(* IEC 61131-3 sources: Lasal/CPU_5344_V01/Class/CtrlCheckMachineReady, 1 file *)

(* ---- CtrlCheckMachineReady.st ---- *)
(*!
<Class
	Name               = "CtrlCheckMachineReady"
	Revision           = "0.1"
	RealtimeTask       = "false"
	CyclicTask         = "true"
	DefCyclictime      = "50 ms"
	BackgroundTask     = "false"
	Sigmatek           = "false"
	OSInterface        = "false"
	HighPriority       = "false"
	Automatic          = "false"
	UpdateMode         = "Prescan"
	SharedCommandTable = "true"
	Objectsize         = "(570,120)">
	<Channels>
		<Server Name="AlarmActiefCommon" Visualized="true" Initialize="false" WriteProtected="false" Retentive="false"/>
		<Server Name="AlarmActiefSafety" Visualized="true" Initialize="false" WriteProtected="false" Retentive="false"/>
		<Server Name="AlarmLubr" Visualized="true" Initialize="false" WriteProtected="false" Retentive="false"/>
		<Server Name="ClassSvr" Visualized="false" Initialize="false" WriteProtected="true" Retentive="false"/>
		<Server Name="ErrorNrCommon" Visualized="true" Initialize="false" WriteProtected="false" Retentive="false"/>
		<Server Name="ErrorNrLubr" Visualized="true" Initialize="false" WriteProtected="false" Retentive="false"/>
		<Server Name="ErrorNrSafety" Visualized="true" Initialize="false" WriteProtected="false" Retentive="false"/>
		<Server Name="ResetAlarms" Visualized="false" Initialize="false" WriteProtected="false" Retentive="false"/>
		<Server Name="result" Class="Logic_Or_2" Visualized="true" Remotely="true" Initialize="false" WriteProtected="true" Retentive="false" Comment="result of logic operation"/>
		<Server Name="sStartUpTime" Visualized="false" Initialize="true" DefValue="10000" WriteProtected="true" Retentive="false"/>
		<Server Name="Status_Controlcurrent" Visualized="false" Initialize="false" WriteProtected="false" Retentive="false"/>
		<Server Name="Status_SafeCompleet" Visualized="false" Initialize="false" WriteProtected="false" Retentive="false"/>
		<Client Name="_AlarmCommon" Required="true" Internal="true"/>
		<Client Name="_AlarmLubr" Required="true" Internal="true"/>
		<Client Name="_AlarmSafety" Required="true" Internal="true"/>
		<Client Name="iBlink" Required="true" Internal="false"/>
		<Client Name="iBTBs" Required="false" Internal="false"/>
		<Client Name="iControlCurrent" Required="true" Internal="false"/>
		<Client Name="iEmergencyStops" Required="false" Internal="false"/>
		<Client Name="iIsafeCompleet" Required="true" Internal="false"/>
		<Client Name="iLuchtdrukOK" Required="false" Internal="false"/>
		<Client Name="iNrLubrs" Required="false" Internal="false"/>
		<Client Name="iSimulateMode" Required="false" Internal="false"/>
		<Client Name="iSmeerSystemenLeeg" Required="false" Internal="false"/>
		<Client Name="iStatusCanComm" Required="true" Internal="false" DefValue="1"/>
		<Client Name="iStuurstroomIn" Required="false" Internal="false"/>
		<Client Name="iThermUits" Required="false" Internal="false"/>
		<Client Name="Logic_Or_23" Required="true" Internal="true"/>
		<Client Name="Logic_Or_24" Required="true" Internal="true"/>
		<Client Name="nrBTBinUse" Required="false" Internal="false"/>
		<Client Name="nrEmergencyStops" Required="false" Internal="false"/>
		<Client Name="nrThermUitinUse" Required="false" Internal="false"/>
		<Client Name="oLightControlCurrent" Required="false" Internal="false"/>
		<Client Name="StatusIOlinkComm" Required="false" Internal="false"/>
	</Channels>
	<RevDoku>
		<Owner/>
		<Dokumentation Revision="0.1" Date="2021-02-09" Author="JDK&#13;&#10;" Company="Dulst" Description="Add lub alarms&#13;&#10;"/>
	</RevDoku>
	<Network Name="CtrlCheckMachineReady">
		<!-- List of Components in this network -->
		<Components>
			<Object
				Name           = "_AlarmCommon"
				Class          = "_AlarmX3ParaDer"
				Position       = "(600,1110)"
				Visualized     = "true"
				Remotely       = "true"
				BackgroundTime = "100 ms">
				<Channels>
					<Server Name="AlarmActief"/>
					<Server Name="ClassSvr"/>
					<Server Name="ErrorNr"/>
					<Client Name="Acknow"/>
					<Client Name="Config" Value="0"/>
					<Client Name="Group"/>
					<Client Name="Para1"/>
					<Client Name="Para2"/>
					<Client Name="Para3"/>
				</Channels>
			</Object>
			<Object
				Name           = "_AlarmLubr"
				Class          = "_AlarmX3ParaDer"
				Position       = "(630,2100)"
				Visualized     = "true"
				Remotely       = "true"
				BackgroundTime = "100 ms">
				<Channels>
					<Server Name="AlarmActief"/>
					<Server Name="ClassSvr"/>
					<Server Name="ErrorNr"/>
					<Client Name="Acknow"/>
					<Client Name="Config" Value="0"/>
					<Client Name="Group"/>
					<Client Name="Para1"/>
					<Client Name="Para2"/>
					<Client Name="Para3"/>
				</Channels>
			</Object>
			<Object
				Name           = "_AlarmSafety"
				Class          = "_AlarmX3ParaDer"
				Position       = "(600,1620)"
				Visualized     = "true"
				Remotely       = "true"
				BackgroundTime = "100 ms">
				<Channels>
					<Server Name="AlarmActief"/>
					<Server Name="ClassSvr"/>
					<Server Name="ErrorNr"/>
					<Client Name="Acknow"/>
					<Client Name="Config" Value="0"/>
					<Client Name="Group"/>
					<Client Name="Para1"/>
					<Client Name="Para2"/>
					<Client Name="Para3"/>
				</Channels>
			</Object>
			<Object
				Name       = "Logic_Or_23"
				Class      = "Logic_Or_2"
				Position   = "(1530,2310)"
				Visualized = "true"
				Remotely   = "true">
				<Channels>
					<Server Name="Result"/>
					<Client Name="Op1"/>
					<Client Name="Op2"/>
				</Channels>
			</Object>
			<Object
				Name       = "Logic_Or_24"
				Class      = "Logic_Or_2"
				Position   = "(1410,1950)"
				Visualized = "true"
				Remotely   = "true">
				<Channels>
					<Server Name="Result"/>
					<Client Name="Op1"/>
					<Client Name="Op2"/>
				</Channels>
			</Object>
		</Components>
		<Comments>
		</Comments>
		<!-- List of Connections in this network -->
		<Connections>
			<Connection Source="this._AlarmLubr" Destination="_AlarmLubr.ClassSvr"/>
			<Connection Source="this._AlarmCommon" Destination="_AlarmCommon.ClassSvr"/>
			<Connection Source="this.AlarmActiefCommon" Destination="_AlarmCommon.AlarmActief" Vertices="(2002,450),(916,1260),"/>
			<Connection Source="this.ErrorNrCommon" Destination="_AlarmCommon.ErrorNr" Vertices="(2002,630),(916,1320),"/>
			<Connection Source="this._AlarmSafety" Destination="_AlarmSafety.ClassSvr"/>
			<Connection Source="this.AlarmActiefSafety" Destination="_AlarmSafety.AlarmActief" Vertices="(2002,510),(916,1770),"/>
			<Connection Source="this.ErrorNrSafety" Destination="_AlarmSafety.ErrorNr" Vertices="(2002,690),(916,1830),"/>
			<Connection Source="this.AlarmLubr" Destination="_AlarmLubr.AlarmActief" Vertices="(2002,570),(946,2250),"/>
			<Connection Source="this.ErrorNrLubr" Destination="_AlarmLubr.ErrorNr" Vertices="(2002,750),(946,2310),"/>
			<Connection Source="this.Logic_Or_23" Destination="Logic_Or_23.Result"/>
			<Connection Source="this.Logic_Or_24" Destination="Logic_Or_24.Result"/>
			<Connection Source="Logic_Or_24.Op1" Destination="_AlarmCommon.AlarmActief" Vertices="(1410,2040),(916,1260),"/>
			<Connection Source="Logic_Or_24.Op2" Destination="_AlarmSafety.AlarmActief" Vertices="(1410,2100),(916,1770),"/>
			<Connection Source="Logic_Or_23.Op2" Destination="_AlarmLubr.AlarmActief" Vertices="(1530,2460),(946,2250),"/>
			<Connection Source="Logic_Or_23.Op1" Destination="Logic_Or_24.Result" Vertices="(1530,2400),(1710,2040),"/>
			<Connection Source="this.result" Destination="Logic_Or_23.Result" Vertices="(2002,870),(1830,2400),"/>
		</Connections>
		<!-- Headerfiles -->
		<Options>
		</Options>
	</Network>
</Class>
*)
CtrlCheckMachineReady : CLASS
  //Servers:
	ClassSvr 	: SvrChCmd_DINT;
	Status_SafeCompleet 	: SvrCh_DINT;
	Status_Controlcurrent 	: SvrCh_DINT;
	ResetAlarms 	: SvrCh_DINT;
	AlarmActiefCommon 	: SvrCh_DINT;
	AlarmActiefSafety 	: SvrCh_DINT;
	AlarmLubr 	: SvrCh_DINT;
	ErrorNrCommon 	: SvrCh_DINT;
	ErrorNrSafety 	: SvrCh_DINT;
	ErrorNrLubr 	: SvrCh_DINT;
	sStartUpTime 	: SvrCh_UDINT;
	result 	: SvrChCmd_DINT;
  //Clients:
	StatusIOlinkComm 	: CltCh_DINT;
	iStatusCanComm 	: CltCh_DINT;
	iStuurstroomIn 	: CltCh_DINT;
	iBTBs 	: CltChCmd_Lees10Ingangenin;
	nrBTBinUse 	: CltCh_DINT;
	iThermUits 	: CltChCmd_Lees10Ingangenin;
	nrThermUitinUse 	: CltCh_DINT;
	iSmeerSystemenLeeg 	: CltCh_DINT;
	iLuchtdrukOK 	: CltCh_DINT;
	iEmergencyStops 	: CltChCmd_Lees10Ingangenin;
	nrEmergencyStops 	: CltCh_DINT;
	oLightControlCurrent 	: CltCh_DINT;
	iSimulateMode 	: CltCh_eSimuState;
	iIsafeCompleet 	: CltCh_DINT;
	iControlCurrent 	: CltCh_DINT;
	iBlink 	: CltCh_DINT;
	iNrLubrs 	: CltCh_DINT;
	_AlarmCommon 	: CltChCmd__AlarmX3ParaDer;
	_AlarmSafety 	: CltChCmd__AlarmX3ParaDer;
	_AlarmLubr 	: CltChCmd__AlarmX3ParaDer;
	Logic_Or_23 	: CltChCmd_Logic_Or_2;
	Logic_Or_24 	: CltChCmd_Logic_Or_2;
  //Variables:
		i 	: DINT;
		ii 	: DINT;
		tmp 	: DINT;
		Status_OldErrorNr 	: DINT;
		tmpErrorNrCommon 	: DINT;
		tmpErrorNrSafety 	: DINT;
		tmpErrorLubr 	: DINT;
  //Functions:

	FUNCTION VIRTUAL GLOBAL CyWork
		VAR_INPUT
			EAX 	: UDINT;
		END_VAR
		VAR_OUTPUT
			state (EAX) 	: UDINT;
		END_VAR;

	FUNCTION CheckNr
		VAR_INPUT
			nr 	: DINT;
			aantaltoread 	: DINT;
			offset 	: DINT;
		END_VAR
		VAR_OUTPUT
			HighNr 	: DINT;
		END_VAR;

	FUNCTION CheckStStrBTBenTherm;

	FUNCTION PreScan;

	FUNCTION CheckSmeerSysteem;

	FUNCTION giveAlarmCommon
		VAR_INPUT
			errorNr 	: DINT;
		END_VAR;

	FUNCTION giveAlarmSafety
		VAR_INPUT
			errorNr 	: DINT;
		END_VAR;

	FUNCTION VIRTUAL GLOBAL ResetAlarms::Write
		VAR_INPUT
			input (EAX) 	: DINT;
		END_VAR
		VAR_OUTPUT
			result (EAX) 	: DINT;
		END_VAR;

	FUNCTION VIRTUAL GLOBAL AlarmActiefCommon::Read
		VAR_OUTPUT
			output (EAX) 	: DINT;
		END_VAR;

	FUNCTION VIRTUAL GLOBAL AlarmActiefCommon::Write
		VAR_INPUT
			input (EAX) 	: DINT;
		END_VAR
		VAR_OUTPUT
			result (EAX) 	: DINT;
		END_VAR;

	FUNCTION VIRTUAL GLOBAL AlarmActiefSafety::Read
		VAR_OUTPUT
			output (EAX) 	: DINT;
		END_VAR;

	FUNCTION VIRTUAL GLOBAL AlarmActiefSafety::Write
		VAR_INPUT
			input (EAX) 	: DINT;
		END_VAR
		VAR_OUTPUT
			result (EAX) 	: DINT;
		END_VAR;

	FUNCTION VIRTUAL GLOBAL AlarmLubr::Read
		VAR_OUTPUT
			output (EAX) 	: DINT;
		END_VAR;

	FUNCTION VIRTUAL GLOBAL AlarmLubr::Write
		VAR_INPUT
			input (EAX) 	: DINT;
		END_VAR
		VAR_OUTPUT
			result (EAX) 	: DINT;
		END_VAR;

	FUNCTION VIRTUAL GLOBAL ErrorNrCommon::Read
		VAR_OUTPUT
			output (EAX) 	: DINT;
		END_VAR;

	FUNCTION VIRTUAL GLOBAL ErrorNrCommon::Write
		VAR_INPUT
			input (EAX) 	: DINT;
		END_VAR
		VAR_OUTPUT
			result (EAX) 	: DINT;
		END_VAR;

	FUNCTION VIRTUAL GLOBAL ErrorNrSafety::Read
		VAR_OUTPUT
			output (EAX) 	: DINT;
		END_VAR;

	FUNCTION VIRTUAL GLOBAL ErrorNrSafety::Write
		VAR_INPUT
			input (EAX) 	: DINT;
		END_VAR
		VAR_OUTPUT
			result (EAX) 	: DINT;
		END_VAR;

	FUNCTION VIRTUAL GLOBAL ErrorNrLubr::Read
		VAR_OUTPUT
			output (EAX) 	: DINT;
		END_VAR;

	FUNCTION VIRTUAL GLOBAL ErrorNrLubr::Write
		VAR_INPUT
			input (EAX) 	: DINT;
		END_VAR
		VAR_OUTPUT
			result (EAX) 	: DINT;
		END_VAR;

	FUNCTION VIRTUAL GLOBAL result::Read
		VAR_OUTPUT
			output (EAX) 	: DINT;
		END_VAR;
  //Tables:
	FUNCTION @STD
		VAR_OUTPUT
			ret_code	: CONFSTATES;
		END_VAR;
	FUNCTION GLOBAL TAB @CT_;
END_CLASS;

#pragma using _AlarmX3ParaDer
#pragma using Logic_Or_2
#pragma usingLtd Lees10Ingangenin

// JdK 22-7-2019: CtrlCheckMachineReady, copied from project 4090
// goal of this fb is to check if every needed input is there, and give an alarm if it isn't

// changed so we can use it for the different sections, signals can be connected to the general check machine ready fb,
// or to the section check machine ready fb, in the last case the signals from the general are also read in, and should
// be ok before signals out are given ok, but there are no alarms given for it

// this class need to be updated some time, but for now we just use it

FUNCTION CtrlCheckMachineReady::CheckStStrBTBenTherm

//errornrs := 1 geen stuurstroom
//            2 geen assenstroom
//            3 tm 12 btb's missen
//            13 tm 22 therms uit missen
//            23 tm 32 luchtdruk te laag
//            33 iSafe weggevallen tijdens productie, reset alarms vereist
//            34 io link niet Ok
//            35 can com niet Ok

// 60 = smeer

  tmpErrorNrCommon := 0;
  if StatusIOlinkComm = 1 & iStatusCanComm = 1 then
    if iStuurstroomIn = 1 then
      //if iLoopwagenstroomIn = 1 then
        tmpErrorNrCommon := CheckNr(nr:=iBTBs, aantaltoread:=nrBTBinUse, offset:=2);
        if tmpErrorNrCommon = 0 then
          tmpErrorNrCommon := CheckNr(nr:=iThermUits, aantaltoread:=nrThermUitinUse, offset:=12);
          if tmpErrorNrCommon = 0 & iLuchtdrukOK = 0 then
            tmpErrorNrCommon := 23;
          end_if;
        end_if;
    elsif tmpErrorNrCommon <> 1 then
      tmpErrorNrCommon := 1;
    end_if;
  elsif StatusIOlinkComm = 0 then
    tmpErrorNrCommon := 34;
  elsif iStatusCanComm = 0 then
    tmpErrorNrCommon := 35;
  end_if;

  if tmpErrorNrCommon = 0 & Status_OldErrorNr <> 2 & Status_OldErrorNr > 0 & Status_OldErrorNr <> 33 & _AlarmCommon.ErrorNr<> 33  then
    _AlarmCommon.AlarmActief.Write(input:=0);
    giveAlarmCommon(errorNr:=33); //deze wordt pas nul bij reset alarms, dan wordt namelijk olderroralgemeen op nul gezet en verdwijnt deze dus
  elsif (tmpErrorNrCommon <> Status_OldErrorNr | (_AlarmCommon.AlarmActief = 0 & tmpErrorNrCommon > 0) ) & Status_OldErrorNr <> 33 & ops.tAbsolute > sStartUpTime  then //don't give alarms during start up
    giveAlarmCommon(errorNr:=tmpErrorNrCommon);
    Status_OldErrorNr := tmpErrorNrCommon;
  end_if;

  if (tmpErrorNrCommon = 0 | iSimulateMode = allSimu) & iIsafeCompleet=1  then
    Status_SafeCompleet := 1;
  else
    Status_SafeCompleet := 0;
  end_if;

  // alarms safety
  oLightControlCurrent := 0;
  iBlink:= iBlink.Read();
  tmpErrorNrSafety := CheckNr(nr:=iEmergencyStops, aantaltoread:=nrEmergencyStops, offset:=0);
  if tmpErrorNrSafety<>0 then
    if ops.tAbsolute > sStartUpTime then //don't give alarms during start up
      giveAlarmSafety(errorNr:=tmpErrorNrSafety);
    end_if;
  else
    _AlarmSafety.ErrorNr := 0; //if em stops are ok, reset alarm
    _AlarmSafety.AlarmActief.Write(input:=0);
    //if iIsafeCompleet= 1 then
      // no alarms
  //    if iAllEmButtons = 0 then
  //      oLightControlCurrent := 0; //one of the em buttons somewhere else is false, so dont flash the light
      (*els*)
      if iStuurstroomIn = 0 then
        // no emergencystops and no control current, turn on light
        oLightControlCurrent := 2;    //JdK 14-10-2020 special because we need to make a difference between two cc zones with one light
      else
        oLightControlCurrent := 1;
      end_if;
    //end_if;
  end_if;
  oLightControlCurrent.Write(input:=oLightControlCurrent);

END_FUNCTION

FUNCTION VIRTUAL GLOBAL CtrlCheckMachineReady::CyWork
	VAR_INPUT
		EAX 	: UDINT;
	END_VAR
	VAR_OUTPUT
		state (EAX) 	: UDINT;
	END_VAR

  PreScan();
  CheckStStrBTBenTherm();
  CheckSmeerSysteem();

	state := READY;

END_FUNCTION

FUNCTION CtrlCheckMachineReady::PreScan
  iSimulateMode := iSimulateMode.Read();
  iStuurstroomIn := iStuurstroomIn.Read();
  Status_Controlcurrent := (iStuurstroomIn | iSimulateMode = allSimu) & iControlCurrent;
  iBTBs := iBTBs.Read(); // we wait two seconds to give time to startup comm
  nrBTBinUse := nrBTBinUse.Read();
  iThermUits := iThermUits.Read();
  nrThermUitinUse := nrThermUitinUse.Read();
  iEmergencyStops := iEmergencyStops.Read();
  iSmeerSystemenLeeg := iSmeerSystemenLeeg.Read();
  iLuchtdrukOK := iLuchtdrukOK.Read() ;
  iStatusCanComm := iStatusCanComm.Read();
  StatusIOlinkComm := StatusIOlinkComm.Read();

  iIsafeCompleet:=iIsafeCompleet.Read();
  iControlCurrent:=iControlCurrent.Read();

END_FUNCTION

FUNCTION CtrlCheckMachineReady::CheckSmeerSysteem

//errors gelijk aan volgorde aansluiten
  iNrLubrs:=iNrLubrs.Read();
  tmpErrorLubr:= CheckNr(nr:=iSmeerSystemenLeeg, aantaltoread:=iNrLubrs, offset:=0);
  if tmpErrorLubr <> _AlarmLubr.ErrorNr then
    _AlarmLubr.ErrorNr.Write(input:=tmpErrorLubr);
    _AlarmLubr.AlarmActief.Write(input:=tmpErrorLubr<>0);
  end_if;

END_FUNCTION

FUNCTION VIRTUAL GLOBAL CtrlCheckMachineReady::ResetAlarms::Write
	VAR_INPUT
		input (EAX) 	: DINT;
	END_VAR
	VAR_OUTPUT
		result (EAX) 	: DINT;
	END_VAR

	ResetAlarms := input;

  Status_OldErrorNr := 0;
  _AlarmCommon.ErrorNr := 0;
  _AlarmCommon.AlarmActief.Write(input:=0);

  _AlarmSafety.ErrorNr := 0;
  _AlarmSafety.AlarmActief.Write(input:=0);
	result := ResetAlarms;

END_FUNCTION

FUNCTION CtrlCheckMachineReady::CheckNr
	VAR_INPUT
		nr 	: DINT;
		aantaltoread 	: DINT;
		offset 	: DINT;
	END_VAR
	VAR_OUTPUT
		HighNr 	: DINT;
	END_VAR

  HighNr := 0;
  for i:= 1 to aantaltoread do
    tmp := nr;
    for ii := 2 to i do
      tmp := tmp/10;
    end_for;
    if tmp mod 10 = 0 then
      HighNr := i + offset;
      exit;
    end_if;
  end_for;

END_FUNCTION

FUNCTION VIRTUAL GLOBAL CtrlCheckMachineReady::AlarmActiefCommon::Read
	VAR_OUTPUT
		output (EAX) 	: DINT;
	END_VAR

	AlarmActiefCommon := _AlarmCommon.AlarmActief.Read();
	output := AlarmActiefCommon;

END_FUNCTION

FUNCTION VIRTUAL GLOBAL CtrlCheckMachineReady::AlarmActiefCommon::Write
	VAR_INPUT
		input (EAX) 	: DINT;
	END_VAR
	VAR_OUTPUT
		result (EAX) 	: DINT;
	END_VAR

	AlarmActiefCommon := input;
	result := (_AlarmCommon.AlarmActief.Write(AlarmActiefCommon))$DINT;

END_FUNCTION

FUNCTION VIRTUAL GLOBAL CtrlCheckMachineReady::AlarmActiefSafety::Read
	VAR_OUTPUT
		output (EAX) 	: DINT;
	END_VAR

	AlarmActiefSafety := _AlarmSafety.AlarmActief.Read();
	output := AlarmActiefSafety;

END_FUNCTION

FUNCTION VIRTUAL GLOBAL CtrlCheckMachineReady::AlarmActiefSafety::Write
	VAR_INPUT
		input (EAX) 	: DINT;
	END_VAR
	VAR_OUTPUT
		result (EAX) 	: DINT;
	END_VAR

	AlarmActiefSafety := input;
	result := (_AlarmSafety.AlarmActief.Write(AlarmActiefSafety))$DINT;

END_FUNCTION

FUNCTION VIRTUAL GLOBAL CtrlCheckMachineReady::ErrorNrCommon::Read
	VAR_OUTPUT
		output (EAX) 	: DINT;
	END_VAR

	ErrorNrCommon := _AlarmCommon.ErrorNr.Read();
	output := ErrorNrCommon;

END_FUNCTION

FUNCTION VIRTUAL GLOBAL CtrlCheckMachineReady::ErrorNrCommon::Write
	VAR_INPUT
		input (EAX) 	: DINT;
	END_VAR
	VAR_OUTPUT
		result (EAX) 	: DINT;
	END_VAR

	ErrorNrCommon := input;
	result := (_AlarmCommon.ErrorNr.Write(ErrorNrCommon))$DINT;

END_FUNCTION

FUNCTION VIRTUAL GLOBAL CtrlCheckMachineReady::ErrorNrSafety::Read
	VAR_OUTPUT
		output (EAX) 	: DINT;
	END_VAR

	ErrorNrSafety := _AlarmSafety.ErrorNr.Read();
	output := ErrorNrSafety;

END_FUNCTION

FUNCTION VIRTUAL GLOBAL CtrlCheckMachineReady::ErrorNrSafety::Write
	VAR_INPUT
		input (EAX) 	: DINT;
	END_VAR
	VAR_OUTPUT
		result (EAX) 	: DINT;
	END_VAR

	ErrorNrSafety := input;
	result := (_AlarmSafety.ErrorNr.Write(ErrorNrSafety))$DINT;

END_FUNCTION

FUNCTION CtrlCheckMachineReady::giveAlarmCommon
	VAR_INPUT
		errorNr 	: DINT;
	END_VAR

  IF _AlarmCommon.AlarmActief=0 | errorNr<>_AlarmCommon.ErrorNr THEN
    _AlarmCommon.ErrorNr.Write(input:=errorNr);
    _AlarmCommon.AlarmActief.Write(input:=1);
  END_IF;

END_FUNCTION

FUNCTION CtrlCheckMachineReady::giveAlarmSafety
	VAR_INPUT
		errorNr 	: DINT;
	END_VAR

  IF _AlarmSafety.AlarmActief=0 | errorNr <> _AlarmSafety.ErrorNr THEN
    _AlarmSafety.ErrorNr.Write(input:=errorNr);
    _AlarmSafety.AlarmActief.Write(input:=1);
  END_IF;

END_FUNCTION

FUNCTION VIRTUAL GLOBAL CtrlCheckMachineReady::AlarmLubr::Read
	VAR_OUTPUT
		output (EAX) 	: DINT;
	END_VAR

	AlarmLubr := _AlarmLubr.AlarmActief.Read();
	output := AlarmLubr;

END_FUNCTION

FUNCTION VIRTUAL GLOBAL CtrlCheckMachineReady::AlarmLubr::Write
	VAR_INPUT
		input (EAX) 	: DINT;
	END_VAR
	VAR_OUTPUT
		result (EAX) 	: DINT;
	END_VAR

	AlarmLubr := input;
	result := (_AlarmLubr.AlarmActief.Write(AlarmLubr))$DINT;

END_FUNCTION

FUNCTION VIRTUAL GLOBAL CtrlCheckMachineReady::ErrorNrLubr::Read
	VAR_OUTPUT
		output (EAX) 	: DINT;
	END_VAR

	ErrorNrLubr := _AlarmLubr.ErrorNr.Read();
	output := ErrorNrLubr;

END_FUNCTION

FUNCTION VIRTUAL GLOBAL CtrlCheckMachineReady::ErrorNrLubr::Write
	VAR_INPUT
		input (EAX) 	: DINT;
	END_VAR
	VAR_OUTPUT
		result (EAX) 	: DINT;
	END_VAR

	ErrorNrLubr := input;
	result := (_AlarmLubr.ErrorNr.Write(ErrorNrLubr))$DINT;

END_FUNCTION

FUNCTION VIRTUAL GLOBAL CtrlCheckMachineReady::result::Read
	VAR_OUTPUT
		output (EAX) 	: DINT;
	END_VAR

	result := Logic_Or_23.Result.Read();
	output := result;

END_FUNCTION
